// SIMATIC S7-200 SMART project (STEP 7-Micro/WIN SMART), CPU SR30

SYMBOL_TABLE 系统符号
First_Scan_On    SM0.1    // 仅在第一个扫描周期时接通
END_SYMBOL_TABLE

ORGANIZATION_BLOCK MAIN:OB1
TITLE=程序注释
BEGIN
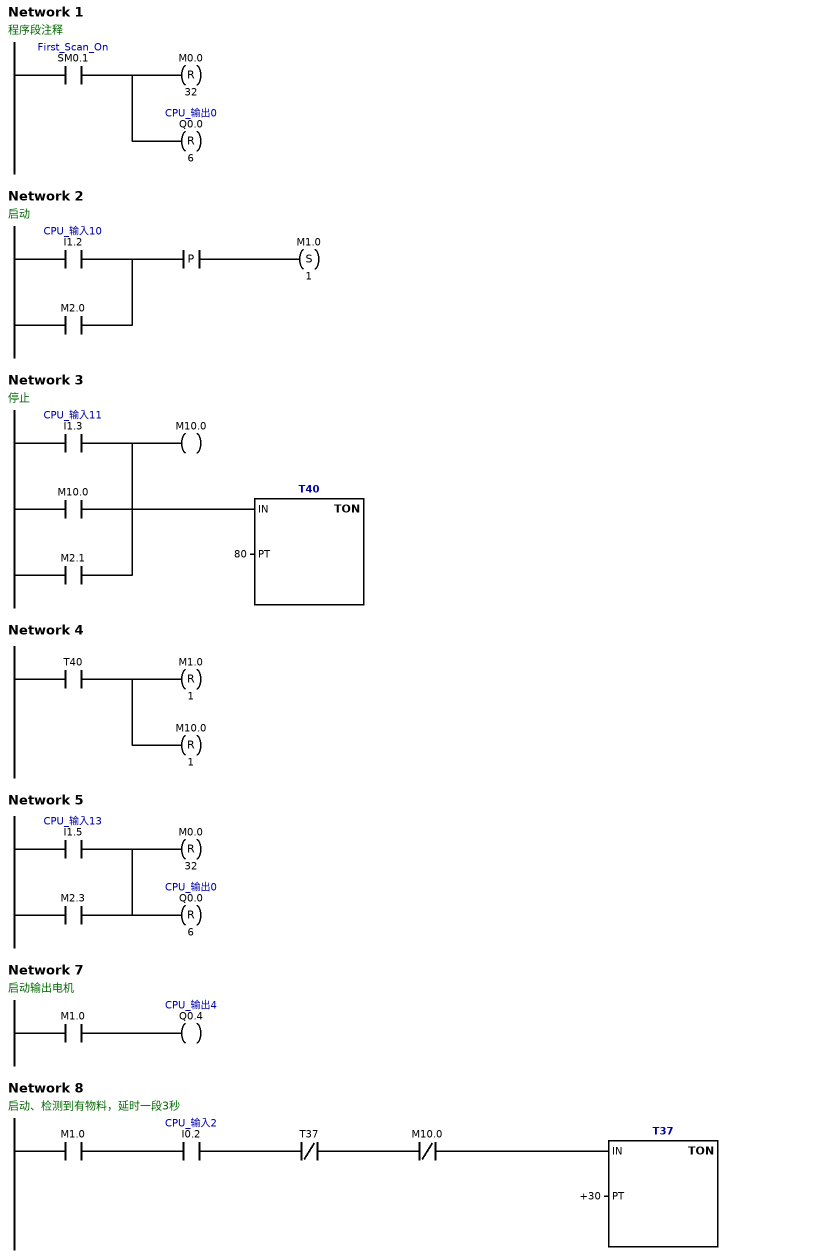
Network 1
// 程序段注释
LD     First_Scan_On:SM0.1
R      M0.0, 32
R      CPU_输出0:Q0.0, 6
Network 2
// 启动
LD     CPU_输入10:I1.2
O      M2.0
EU
S      M1.0, 1
Network 3
// 停止
LD     CPU_输入11:I1.3
O      M10.0
O      M2.1
=      M10.0
TON    T40, 80
Network 4
LD     T40
R      M1.0, 1
R      M10.0, 1
Network 5
LD     CPU_输入13:I1.5
O      M2.3
R      M0.0, 32
R      CPU_输出0:Q0.0, 6
Network 7
// 启动输出电机
LD     M1.0
=      CPU_输出4:Q0.4
Network 8
// 启动、检测到有物料，延时一段3秒
LD     M1.0
A      CPU_输入2:I0.2
AN     T37
AN     M10.0
TON    T37, +30
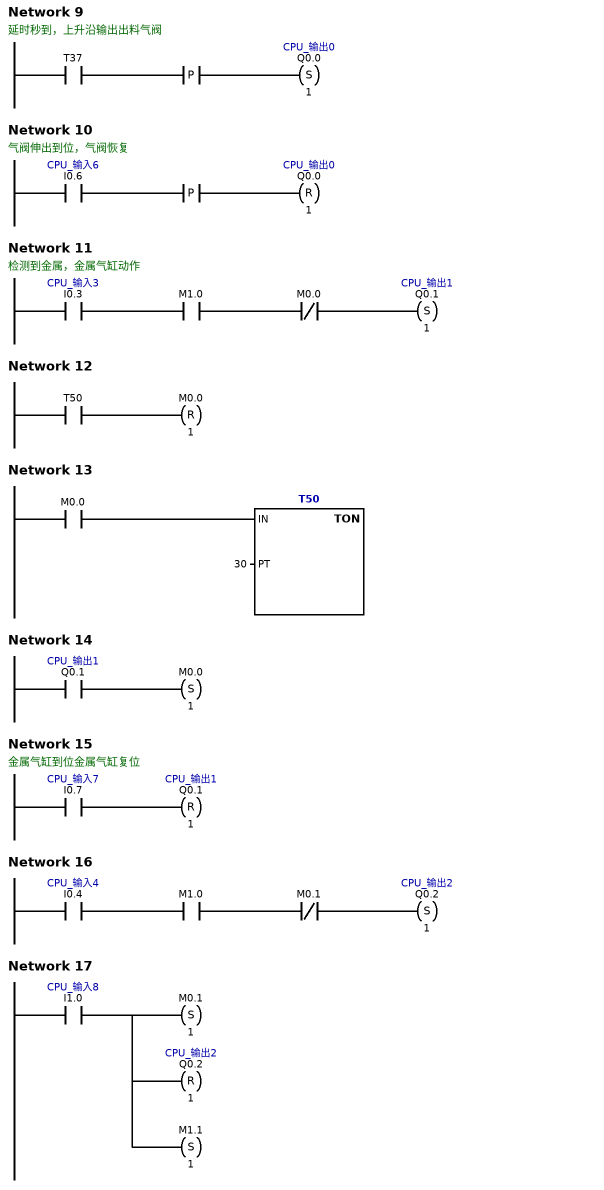
Network 9
// 延时秒到，上升沿输出出料气阀
LD     T37
EU
S      CPU_输出0:Q0.0, 1
Network 10
// 气阀伸出到位，气阀恢复
LD     CPU_输入6:I0.6
EU
R      CPU_输出0:Q0.0, 1
Network 11
// 检测到金属，金属气缸动作
LD     CPU_输入3:I0.3
A      M1.0
AN     M0.0
S      CPU_输出1:Q0.1, 1
Network 12
LD     T50
R      M0.0, 1
Network 13
LD     M0.0
TON    T50, 30
Network 14
LD     CPU_输出1:Q0.1
S      M0.0, 1
Network 15
// 金属气缸到位金属气缸复位
LD     CPU_输入7:I0.7
R      CPU_输出1:Q0.1, 1
Network 16
LD     CPU_输入4:I0.4
A      M1.0
AN     M0.1
S      CPU_输出2:Q0.2, 1
Network 17
LD     CPU_输入8:I1.0
S      M0.1, 1
R      CPU_输出2:Q0.2, 1
S      M1.1, 1
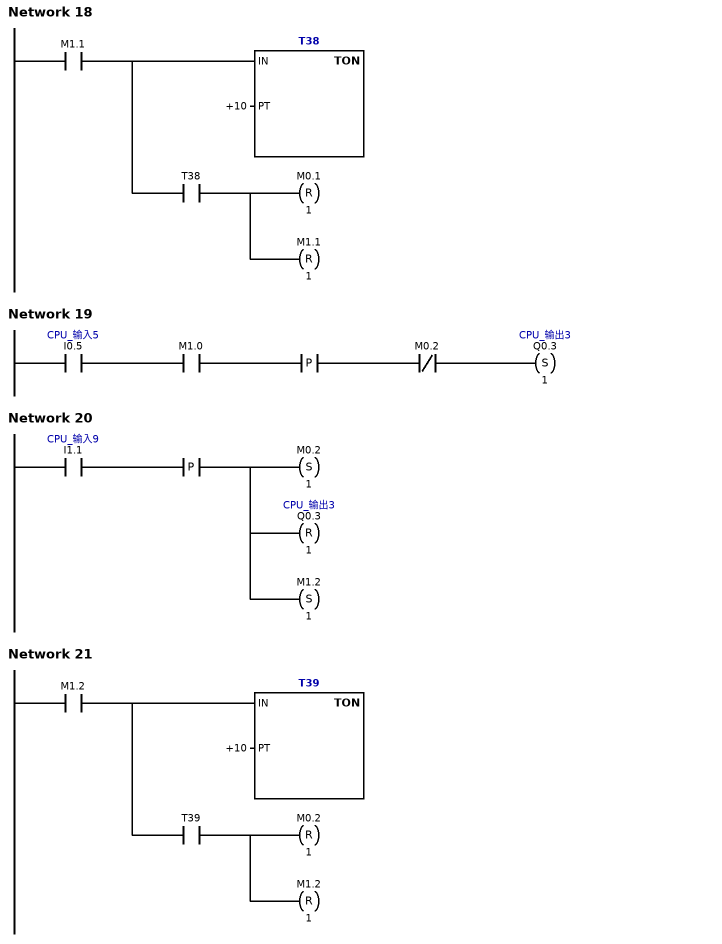
Network 18
LD     M1.1
TON    T38, +10
A      T38
R      M0.1, 1
R      M1.1, 1
Network 19
LD     CPU_输入5:I0.5
A      M1.0
EU
AN     M0.2
S      CPU_输出3:Q0.3, 1
Network 20
LD     CPU_输入9:I1.1
EU
S      M0.2, 1
R      CPU_输出3:Q0.3, 1
S      M1.2, 1
Network 21
LD     M1.2
TON    T39, +10
A      T39
R      M0.2, 1
R      M1.2, 1
END_ORGANIZATION_BLOCK
